{attribute 'pack_mode' := '1'}
    {attribute 'OPC.UA.DA' := '1'}
    {attribute 'OPC.UA.DA.StructuredType' := '1'}
    (*
    ST_RW_RealMemory_HMI_IgnitionExp
    ==================================================
    Generated from Ignition UDT: RW_Real_Memory
    Total tags: 1
    Generated on: 2025-09-15 12:56:43
    *)
    TYPE ST_RW_RealMemory_HMI_IgnitionExp :
    STRUCT
        {attribute 'OPC.UA.DA' := '1'}
        {attribute 'OPC.UA.DA.Description' := '{Description}'}
        // {Description}
        Value : REAL := 0.0;
    END_STRUCT
    END_TYPE

(* stored: Version 1.1.0.1
   DUT ST_RW_RealMemory_HMI_IgnitionExp: Id {ba37d61d-75b8-4ae2-9b6e-062fa4a0890e} *)
